FUNCTION F_CheckAxisGEQ : BOOL
VAR_INPUT
    stMotionStage: ST_MotionStage;
    fQueryValue: LREAL;
END_VAR
VAR
END_VAR


F_CheckAxisGEQ := F_CheckAxis(stMotionStage, 3, fQueryValue);

END_FUNCTION

(* stored: Version 1.1.0.1, ProductVersion 3.1.4022.18
   POU F_CheckAxisGEQ: Id {7634f106-b007-474f-8820-62f9e7a6a689}, SpecialFunc None *)
